# EPICS SNL sequencer program: viocs/si_ps/si_psApp/src/ps_sp_init.stt
program ps_sp_init

int event_proc;
assign event_proc to "EVENT-SIPS-SP-INIT.PROC";

ss ss1 {
    state init {
        when (delay(.5)) {
            event_proc = 1;
            pvPut(event_proc);
        } exit
    }
}
